PROGRAM PRG_11_ScreenButtons
VAR
	TON_CarriageEnable: TON;	
	TON_TurretEnable: TON;
	R_TRIG_0: R_TRIG;
	R_TRIG_1: R_TRIG;
	TON_Horn: TON;
	TON_DriveFast: TON;
	R_TRIG_2: R_TRIG;
	TON_MachineHoming: TON;
	TON_CrossCutPosition: TON;
	TON_AutoCrossCut: TON;
	TON_LeftLimit: TON;
	TON_RightLimit: TON;
	F_TRIG_0: F_TRIG;
	F_TRIG_1: F_TRIG;
	R_TRIG_3: R_TRIG;
	TOF_Teach: TOF;
	F_TRIG_2: F_TRIG;
	TOF_TeachSuccess: TOF;
	TON_DownLimitCaptureReady: TON;
	TON_DownLimitCaptureReady2: TON;

	R_TRIG_4: R_TRIG;
	TOF_CaptureSuccess: TOF;
	TON_BladeCutCountReset: TON;
	TON_DoublePassEnable: TON;
	SR_DoublePass: SR;
	F_TRIG_3: F_TRIG;
	SR_TurretEnableTimeout: SR;
	R_TRIG_5: R_TRIG;
	R_TRIG_6: R_TRIG;
	SR_CarriageEnableTimeout: SR;
	R_TRIG_7: R_TRIG;
	R_TRIG_8: R_TRIG;
	SR_DriveFastTimeout: SR;
	R_TRIG_9: R_TRIG;
	R_TRIG_10: R_TRIG;
	R_TRIG_11: R_TRIG;
	R_TRIG_12: R_TRIG;
	R_TRIG_13: R_TRIG;
	R_TRIG_14: R_TRIG;
	R_TRIG_15: R_TRIG;
	R_TRIG_16: R_TRIG;
	R_TRIG_17: R_TRIG;
	R_TRIG_18: R_TRIG;
	R_TRIG_19: R_TRIG;
	R_TRIG_20: R_TRIG;
END_VAR
VAR // added by the converter: edge detectors and wires of the graphical bodies
    _w1, _w2, _w3 : BOOL;
END_VAR

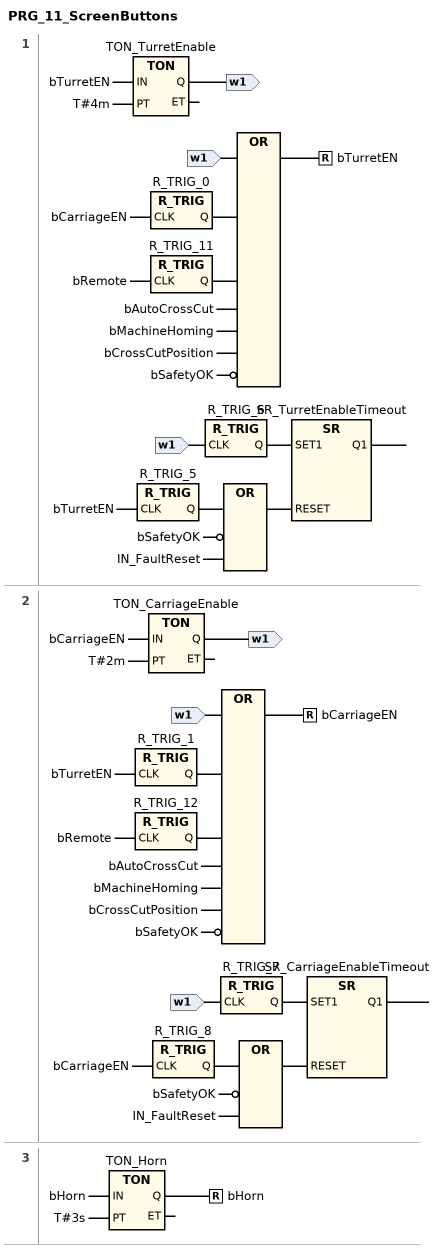
// NETWORK 1
TON_TurretEnable(IN := bTurretEN, PT := T#4m); // TON
R_TRIG_0(CLK := bCarriageEN); // R_TRIG
R_TRIG_11(CLK := bRemote); // R_TRIG
bTurretEN R= TON_TurretEnable.Q OR R_TRIG_0.Q OR R_TRIG_11.Q OR bAutoCrossCut OR bMachineHoming OR bCrossCutPosition OR NOT bSafetyOK;
R_TRIG_6(CLK := TON_TurretEnable.Q); // R_TRIG
R_TRIG_5(CLK := bTurretEN); // R_TRIG
SR_TurretEnableTimeout(SET1 := R_TRIG_6.Q, RESET := R_TRIG_5.Q OR NOT bSafetyOK OR IN_FaultReset); // SR

// NETWORK 2
TON_CarriageEnable(IN := bCarriageEN, PT := T#2m); // TON
R_TRIG_1(CLK := bTurretEN); // R_TRIG
R_TRIG_12(CLK := bRemote); // R_TRIG
bCarriageEN R= TON_CarriageEnable.Q OR R_TRIG_1.Q OR R_TRIG_12.Q OR bAutoCrossCut OR bMachineHoming OR bCrossCutPosition OR NOT bSafetyOK;
R_TRIG_7(CLK := TON_CarriageEnable.Q); // R_TRIG
R_TRIG_8(CLK := bCarriageEN); // R_TRIG
SR_CarriageEnableTimeout(SET1 := R_TRIG_7.Q, RESET := R_TRIG_8.Q OR NOT bSafetyOK OR IN_FaultReset); // SR

// NETWORK 3
TON_Horn(IN := bHorn, PT := T#3s); // TON
bHorn R= TON_Horn.Q;

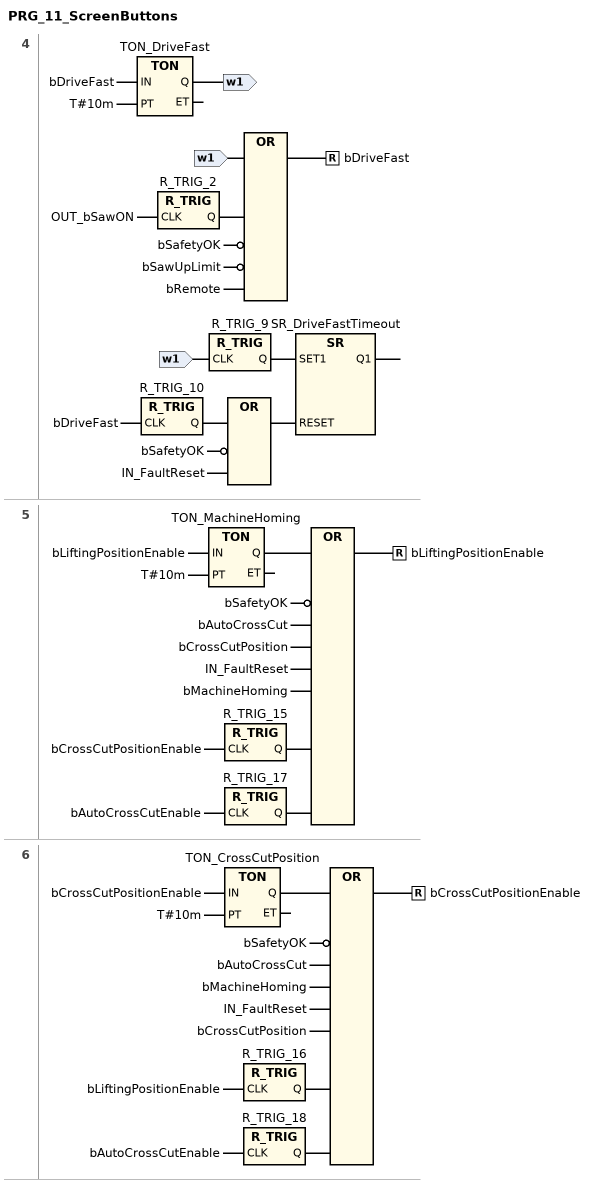
// NETWORK 4
TON_DriveFast(IN := bDriveFast, PT := T#10m); // TON
R_TRIG_2(CLK := OUT_bSawON); // R_TRIG
bDriveFast R= TON_DriveFast.Q OR R_TRIG_2.Q OR NOT bSafetyOK OR NOT bSawUpLimit OR bRemote;
R_TRIG_9(CLK := TON_DriveFast.Q); // R_TRIG
R_TRIG_10(CLK := bDriveFast); // R_TRIG
SR_DriveFastTimeout(SET1 := R_TRIG_9.Q, RESET := R_TRIG_10.Q OR NOT bSafetyOK OR IN_FaultReset); // SR

// NETWORK 5
TON_MachineHoming(IN := bLiftingPositionEnable, PT := T#10m); // TON
R_TRIG_15(CLK := bCrossCutPositionEnable); // R_TRIG
R_TRIG_17(CLK := bAutoCrossCutEnable); // R_TRIG
bLiftingPositionEnable R= TON_MachineHoming.Q OR NOT bSafetyOK OR bAutoCrossCut OR bCrossCutPosition OR IN_FaultReset OR bMachineHoming OR R_TRIG_15.Q OR R_TRIG_17.Q;

// NETWORK 6
TON_CrossCutPosition(IN := bCrossCutPositionEnable, PT := T#10m); // TON
R_TRIG_16(CLK := bLiftingPositionEnable); // R_TRIG
R_TRIG_18(CLK := bAutoCrossCutEnable); // R_TRIG
bCrossCutPositionEnable R= TON_CrossCutPosition.Q OR NOT bSafetyOK OR bAutoCrossCut OR bMachineHoming OR IN_FaultReset OR bCrossCutPosition OR R_TRIG_16.Q OR R_TRIG_18.Q;

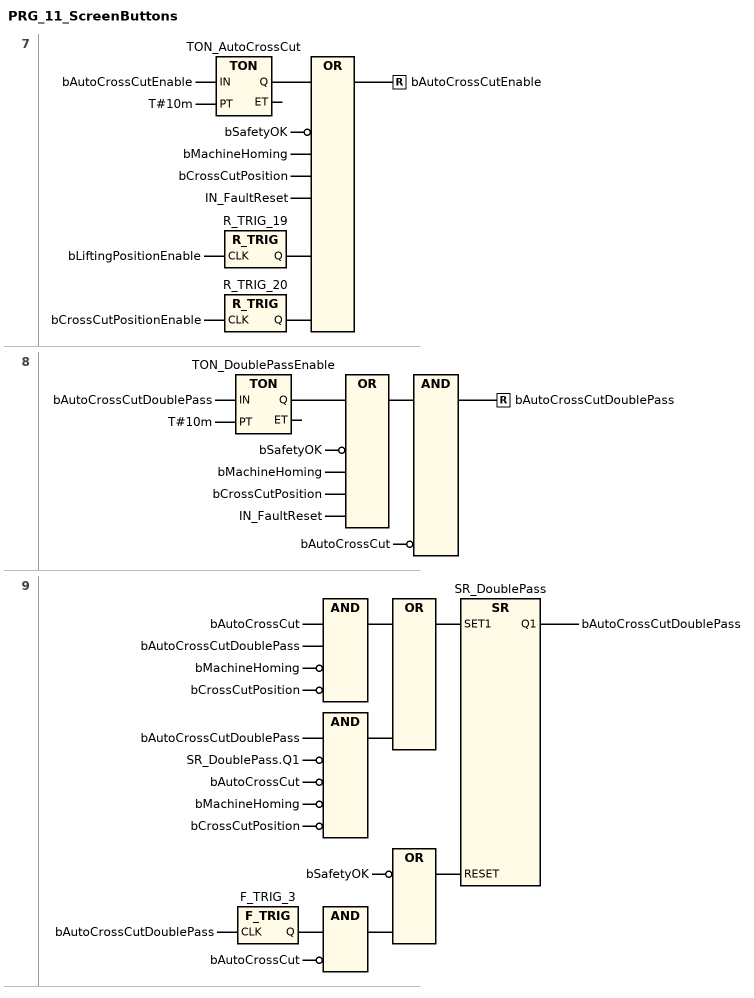
// NETWORK 7
TON_AutoCrossCut(IN := bAutoCrossCutEnable, PT := T#10m); // TON
R_TRIG_19(CLK := bLiftingPositionEnable); // R_TRIG
R_TRIG_20(CLK := bCrossCutPositionEnable); // R_TRIG
bAutoCrossCutEnable R= TON_AutoCrossCut.Q OR NOT bSafetyOK OR bMachineHoming OR bCrossCutPosition OR IN_FaultReset OR R_TRIG_19.Q OR R_TRIG_20.Q;

// NETWORK 8
TON_DoublePassEnable(IN := bAutoCrossCutDoublePass, PT := T#10m); // TON
bAutoCrossCutDoublePass R= (TON_DoublePassEnable.Q OR NOT bSafetyOK OR bMachineHoming OR bCrossCutPosition OR IN_FaultReset) AND NOT bAutoCrossCut;

// NETWORK 9
F_TRIG_3(CLK := bAutoCrossCutDoublePass); // F_TRIG
SR_DoublePass(SET1 := bAutoCrossCut AND bAutoCrossCutDoublePass AND NOT bMachineHoming AND NOT bCrossCutPosition OR bAutoCrossCutDoublePass AND NOT SR_DoublePass.Q1 AND NOT bAutoCrossCut AND NOT bMachineHoming AND NOT bCrossCutPosition, RESET := NOT bSafetyOK OR F_TRIG_3.Q AND NOT bAutoCrossCut); // SR
bAutoCrossCutDoublePass := SR_DoublePass.Q1;

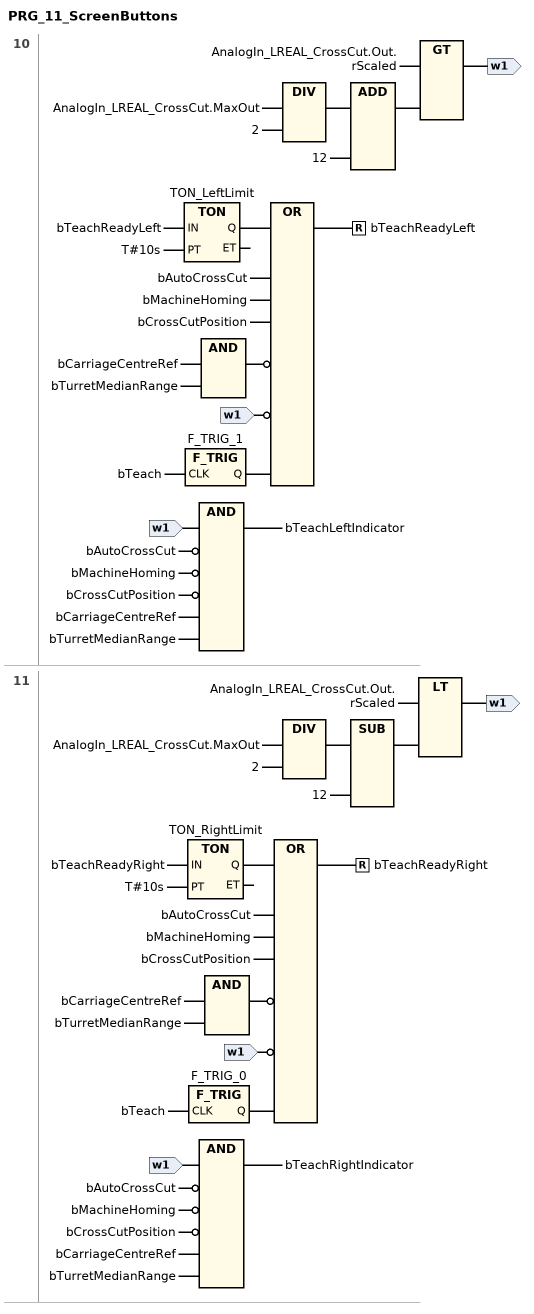
// NETWORK 10
_w1 := AnalogIn_LREAL_CrossCut.Out.rScaled > AnalogIn_LREAL_CrossCut.MaxOut / 2 + 12;
TON_LeftLimit(IN := bTeachReadyLeft, PT := T#10s); // TON
F_TRIG_1(CLK := bTeach); // F_TRIG
bTeachReadyLeft R= TON_LeftLimit.Q OR bAutoCrossCut OR bMachineHoming OR bCrossCutPosition OR NOT (bCarriageCentreRef AND bTurretMedianRange) OR NOT _w1 OR F_TRIG_1.Q;
bTeachLeftIndicator := _w1 AND NOT bAutoCrossCut AND NOT bMachineHoming AND NOT bCrossCutPosition AND bCarriageCentreRef AND bTurretMedianRange;

// NETWORK 11
_w2 := AnalogIn_LREAL_CrossCut.Out.rScaled < AnalogIn_LREAL_CrossCut.MaxOut / 2 - 12;
TON_RightLimit(IN := bTeachReadyRight, PT := T#10s); // TON
F_TRIG_0(CLK := bTeach); // F_TRIG
bTeachReadyRight R= TON_RightLimit.Q OR bAutoCrossCut OR bMachineHoming OR bCrossCutPosition OR NOT (bCarriageCentreRef AND bTurretMedianRange) OR NOT _w2 OR F_TRIG_0.Q;
bTeachRightIndicator := _w2 AND NOT bAutoCrossCut AND NOT bMachineHoming AND NOT bCrossCutPosition AND bCarriageCentreRef AND bTurretMedianRange;

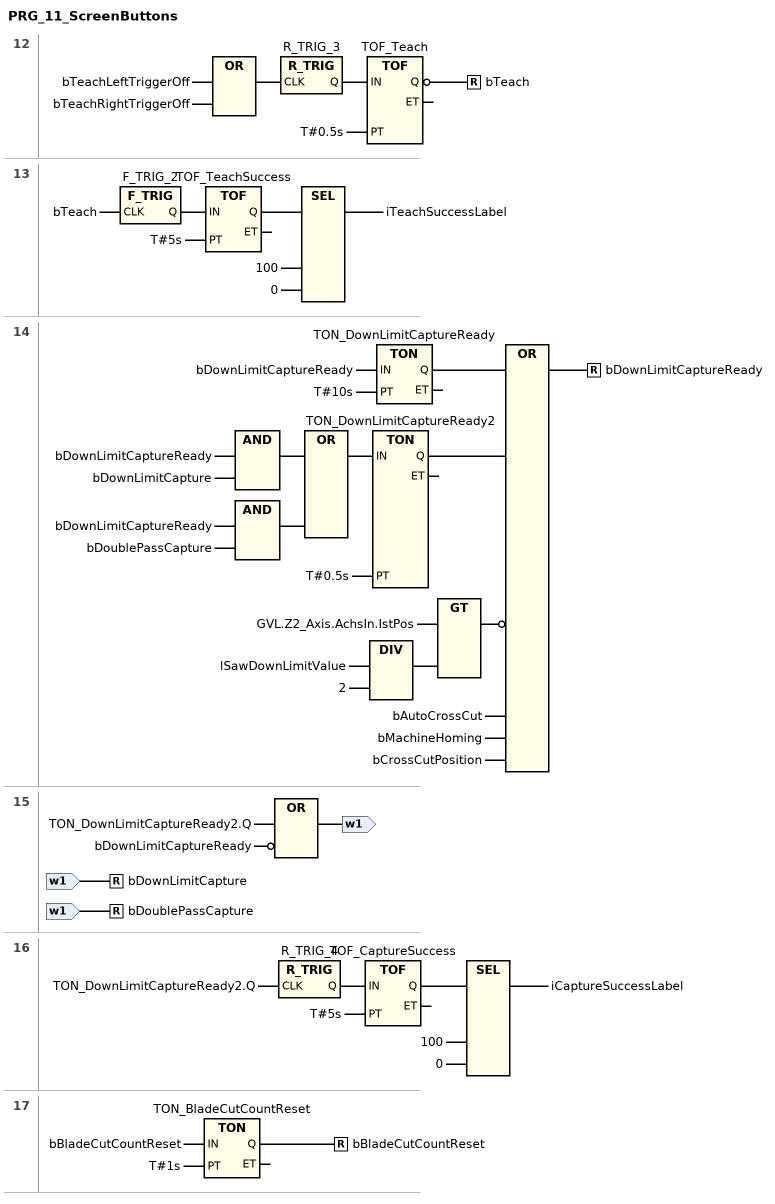
// NETWORK 12
R_TRIG_3(CLK := bTeachLeftTriggerOff OR bTeachRightTriggerOff); // R_TRIG
TOF_Teach(IN := R_TRIG_3.Q, PT := T#0.5s); // TOF
bTeach R= NOT TOF_Teach.Q;

// NETWORK 13
F_TRIG_2(CLK := bTeach); // F_TRIG
TOF_TeachSuccess(IN := F_TRIG_2.Q, PT := T#5s); // TOF
iTeachSuccessLabel := SEL(TOF_TeachSuccess.Q, 100, 0);

// NETWORK 14
TON_DownLimitCaptureReady(IN := bDownLimitCaptureReady, PT := T#10s); // TON
TON_DownLimitCaptureReady2(IN := bDownLimitCaptureReady AND bDownLimitCapture OR bDownLimitCaptureReady AND bDoublePassCapture, PT := T#0.5s); // TON
bDownLimitCaptureReady R= TON_DownLimitCaptureReady.Q OR TON_DownLimitCaptureReady2.Q OR NOT (GVL.Z2_Axis.AchsIn.IstPos > lSawDownLimitValue / 2) OR bAutoCrossCut OR bMachineHoming OR bCrossCutPosition;

// NETWORK 15
_w3 := TON_DownLimitCaptureReady2.Q OR NOT bDownLimitCaptureReady;
bDownLimitCapture R= _w3;
bDoublePassCapture R= _w3;

// NETWORK 16
R_TRIG_4(CLK := TON_DownLimitCaptureReady2.Q); // R_TRIG
TOF_CaptureSuccess(IN := R_TRIG_4.Q, PT := T#5s); // TOF
iCaptureSuccessLabel := SEL(TOF_CaptureSuccess.Q, 100, 0);

// NETWORK 17
TON_BladeCutCountReset(IN := bBladeCutCountReset, PT := T#1s); // TON
bBladeCutCountReset R= TON_BladeCutCountReset.Q;

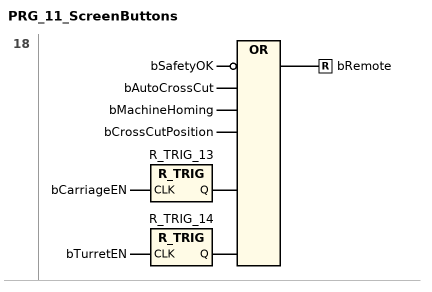
// NETWORK 18
R_TRIG_13(CLK := bCarriageEN); // R_TRIG
R_TRIG_14(CLK := bTurretEN); // R_TRIG
bRemote R= NOT bSafetyOK OR bAutoCrossCut OR bMachineHoming OR bCrossCutPosition OR R_TRIG_13.Q OR R_TRIG_14.Q;

END_PROGRAM

(* stored: Version 1.1.0.1, ProductVersion 3.1.4024.15
   POU PRG_11_ScreenButtons: Id {f1093085-a14a-4abd-bbcd-9bc7142bd274}, SpecialFunc None *)
